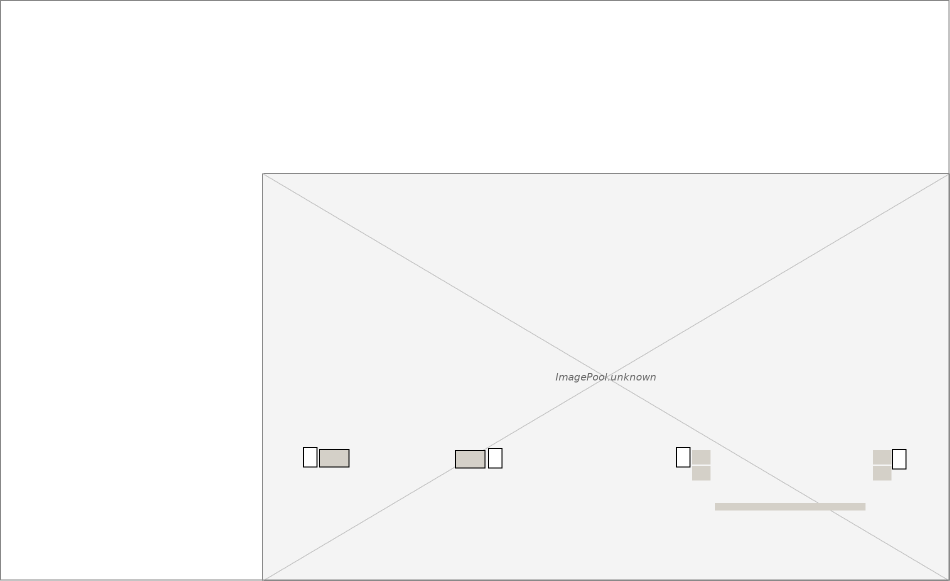
VISUALIZATION Lights  // 950x581
    Image (262,173 688x408), image: ImagePool.unknown
    RoundedRectangle (488,448 14x20), colour toggle: RunTCP.BlinkerLeft
    RoundedRectangle (303,447 14x20), colour toggle: RunTCP.BlinkerRight
    RoundedRectangle (455,450 30x18), colour toggle: RunTCP.LightsFront
    RoundedRectangle (676,447 14x20), colour toggle: RunTCP.BlinkerLeft
    RoundedRectangle (892,449 14x20), colour toggle: RunTCP.BlinkerRight
    RoundedRectangle (319,449 30x18), colour toggle: RunTCP.LightsFront
    RoundedRectangle (692,450 18x14), colour toggle: RunTCP.LightsRear
    RoundedRectangle (692,466 18x14), colour toggle: RunTCP.LightsBrake
    RoundedRectangle (873,450 18x14), colour toggle: RunTCP.LightsRear
    RoundedRectangle (873,466 18x14), colour toggle: RunTCP.LightsBrake
    RoundedRectangle (715,503 150x7), colour toggle: RunTCP.LightsReverse
END_VISUALIZATION

(* stored: Version 1.1.0.1, ProductVersion 3.1.4024.3
   Visu Lights: Id {a493a650-b676-4b8f-b316-5c9c8526622b} *)
